Fanuc KAREL source: kt00906.KL

-- PROVISIONAL review KL for V1013-1; original PC SHA256 d7385ce8c036456bb6209809c6858b061a7a231dcbbc72e77d6aa100c98803c4
-- Incomplete behavior may be omitted. Consult companion uncertainty JSON. Do not deploy.
PROGRAM KT00906
%NOLOCKGROUP
BEGIN
  -- UNRESOLVED_PC offsets 5-31; opcodes 27,27,49,7E,AD,31,4A
  -- UNRESOLVED_PC offsets 36-40; opcodes 7F
END KT00906
